(*

.. <legal notes>

legal notes
=================
| SPDX-FileCopyrightText: © 2026 Oleksandr Tiutyk <trofimich@gmail.com>
| SPDX-License-Identifier: LGPL-3.0-only
| For details check: LGPL-3.0-only_

.. _LGPL-3.0-only: https://www.gnu.org/licenses/lgpl-3.0.en.html

.. </legal notes>

*)

INTERFACE IConfigurableSimulatable EXTENDS ISimulatable

METHOD SetSimulationMode
VAR_INPUT
	value : BOOL;
END_VAR
END_METHOD

END_INTERFACE

(* stored: Version 1.1.0.1
   Itf IConfigurableSimulatable: Id {3effb189-bda6-4e90-acdc-0316c3a2a295}
   Method SetSimulationMode: Id {2ec04501-b180-403d-934c-f7710f1907a0} *)
